FUNCTION_BLOCK GetInstancePath (* Service Interface Function Block Type *)
  (* Description: Copyright (c) 2023 Primetals Technologies Austria GmbH This program and the accompanying materials are made available under the terms of the Eclipse Public License 2.0 which is available at https://www.eclipse.org/legal/epl-2.0/ SPDX-License-Identifier: EPL-2.0 *)
  (* Version 1.0, 2012-12-10, Alois Zoitl, Primetals Technologies Austria GmbH *)
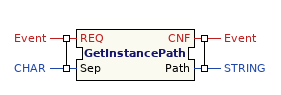
  EVENT_INPUT
    REQ WITH Sep; (* Service Request *)
  END_EVENT
  EVENT_OUTPUT
    CNF WITH Path; (* Confirmation of Requested Service *)
  END_EVENT
  VAR_INPUT
    Sep : CHAR := '/'; (* Separator character for the output path generated by this FB *)
  END_VAR
  VAR_OUTPUT
    Path : STRING; (* Instance path of this FB *)
  END_VAR
  SERVICE APPLICATION/RESOURCE (* Service Interface Function Block Type *)
    SEQUENCE Normal operation
      APPLICATION.REQ(Sep) -> RESOURCE.acquire path information(Sep) -> APPLICATION.CNF(Path);
    END_SEQUENCE
  END_SERVICE
END_FUNCTION_BLOCK
